(* IEC 61131-3 sources: YaoKangDeviceDemo/src/00_Globals, 6 files *)

(* ---- ST_StruHMI.st ---- *)
(*============================================================================
  HMI 线上结构体类型库 —— 寄存器布局契约
  ----------------------------------------------------------------------------
  权威来源：旧工程 InoProShop 变量表导出
    old/结构体/Stru_HMI_new.csv                     （主结构体，AT %MW200）
    old/结构体/Stru_HMI_DeviceInfo_new.csv          （设备信息镜像，AT %MW1000）
    old/结构体/Stru_HMI_DeviceIdentityWrite_new.csv （设备身份维护，AT %MW1010）

  ⚠ 铁律：类型名、字段名、字段顺序、数据类型、数组长度必须与 CSV 完全一致，
     一字不改。BOOL 按位打包、REAL/DINT 偶字对齐由编译器自动完成；
     本工程照抄定义并整体 AT 映射后，布局即与旧工程/HMI 完全相同。
  验收：下载后 InoProShop 变量表中 HMI 的 nBitLen 应 = 11856 bit（741 字，
        D200–D940），与旧工程一致。
==========================================================================*)

(*---------------------------------------------------------------------------
  通用命令：参数块统一操作集（Load/Apply/Save/ResetDefault + 回令）
  出现位置：Condition.ParamCmd / TailTilt.ConfigCmd / 3×Axis.ConfigCmd / HomingParams.Cmd
---------------------------------------------------------------------------*)
TYPE Stru_ConfigCmd :
STRUCT
    iErrorCode      : INT;      // 操作错误
    bLoad           : BOOL;     // 加载：从运行区读到缓冲区
    bApply          : BOOL;     // 应用：缓冲区覆盖运行区
    bSave           : BOOL;     // 保存：运行区写入 Retain
    bResetDefault   : BOOL;     // 恢复工厂默认
    bSuccess        : BOOL;     // 操作成功（PLC→HMI 回令）
    bError          : BOOL;     // 操作失败（只读，PLC→HMI 回令）
    bPad0           : BOOL;     // 填充
    bPad1           : BOOL;     // 对齐填充
END_STRUCT
END_TYPE

(*---------------------------------------------------------------------------
  调理区（Condition）
---------------------------------------------------------------------------*)
TYPE Stru_CondCmd :
STRUCT
    S1_StartProcess     : BOOL;     // 启动流程 (电平，CSV 注释；PLC 侧按 R_TRIG 消费亦安全)
    S2_StartChengJiao   : BOOL;     // 开始成角 (脉冲)
    S3_AllowSignal      : BOOL;     // 确认信号 (脉冲)
    bStop               : BOOL;     // 停止 (脉冲)
    bSignal             : BOOL;     // 脚踏信号 (脉冲/电平)
    bReset              : BOOL;     // 复位错误 (脉冲)
    bPause              : BOOL;     // 暂停
    bResume             : BOOL;     // 恢复
    bSkipAngle          : BOOL;     // 跳过成角 (脉冲, v3.16)
    bPpad               : BOOL[7];  // 填充（字段名照抄 CSV：bPpad）
END_STRUCT
END_TYPE

(* 单轴往复运动参数（SeatTwist / LegAngle / ChestImpact 三处复用） *)
TYPE Stru_ReciprocationSettings :
STRUCT
    arPosition      : REAL[16];    // 各段目标位置
    arVelocity      : REAL[16];    // 各段速度
    rAcc            : REAL;        // 加速度（必须 > 0）
    rDec            : REAL;        // 减速度（必须 > 0）
    rInitialPosition: REAL;        // 初始位置
    rReserved       : REAL;        // 保留
    iVelocityMode   : INT;         // 速度切换模式 0=独立速度 1=统一用 arVelocity[0]
    iCycleModeLen   : INT;         // 方向数组 abCycleMode 有效长度 (1~16)
    iCycleCount     : INT;         // 本轴循环次数，-1=用全局值
    iSignalMode     : INT;         // 本轴信号模式，-1=用全局值，0=点动 1=连动
    iSegmentCount   : INT;         // 运动段数 (1~16)，必须 >0 否则报错 1005
    iPadInt         : INT;         // 对齐填充
    bEnabled        : BOOL;        // 轴使能（FALSE=不参与联动，用于 2 轴场景）
    bOneWay         : BOOL;        // 单向还是多向
    abCycleMode     : BOOL[16];    // 方向数组
    bPad0           : BOOL;        // 填充
    bPad1           : BOOL;        // 对齐填充
END_STRUCT
END_TYPE

TYPE Stru_CondParams :
STRUCT
    SeatTwist       : Stru_ReciprocationSettings;   // 扭腰往复（线上顺序 Seat→Leg→Chest）
    LegAngle        : Stru_ReciprocationSettings;   // 摆腿往复
    ChestImpact     : Stru_ReciprocationSettings;   // 冲击往复
    rPusherPos      : REAL;        // 成角角度（尾板目标角度，度）
    rPusherInitPos   : REAL;        // 尾板初始角度
    diBatchCount    : DINT;        // 完整调理流程重复次数（老化模式）
    diBatchInterval : DINT;        // 批次间隔时间 (ms，老化模式)
    diTotalTimeout  : DINT;        // 总超时 (ms，默认 300000)
    diConfirmTimeout: DINT;        // HMI 等待确认超时 (ms，<=0=禁用)
    iCycleCount     : INT;         // 全局循环次数
    iSignalMode     : INT;         // 全局信号模式 (0=脚踏 1=自动)
END_STRUCT
END_TYPE

TYPE Stru_CondStatus :
STRUCT
    diActRunTime        : DINT;    // 实际运行时间 (ms，含暂停)
    diBatchCurrent      : DINT;    // 已完成批次数（老化）
    diBatchTarget       : DINT;    // 目标批次数（老化）
    diBatchRemainTime   : DINT;    // 批次间隔剩余时间 (ms)
    iPhase              : INT;     // 调理阶段 (0=空闲 1=预备 2=运行 3=成角 9=完成)
    iStep               : INT;     // 当前步骤（阶段内细分）
    iCurrentCycle       : INT;     // 当前循环次数
    iTargetCycles       : INT;     // 目标循环次数
    iErrorCode          : INT;     // 错误码
    iErrorLevel         : INT;     // 错误等级 0=L0 1=L1 2=L2
    iParamError         : INT;     // 参数验证错误码
    iParamErrorAxis     : INT;     // 参数错误所在轴 (1=Chest 2=Leg 3=Seat 4=Tail)
    iParamErrorField    : INT;     // 错误字段索引
    pad_int             : INT;     // 对齐填充
    bRunning            : BOOL;    // 调理进行中
    bDone               : BOOL;    // 调理已完成
    bPaused             : BOOL;    // 暂停中
    bError              : BOOL;    // 错误激活
    bBusy               : BOOL;    // 任意动作进行中
    bWaitingAngle       : BOOL;    // 等待成角
    bHoming             : BOOL;    // 回零中
    bAngleDone          : BOOL;    // 成角已完成
    bWaitingSignal      : BOOL;    // 等待脚踏信号
    bMoving             : BOOL;    // 往复动作中
    bHomeDone           : BOOL;    // 回零完成
    bManualStop         : BOOL;    // 手动停止
    bEmergencyStop      : BOOL;    // 紧急中止
    bParamValid         : BOOL;    // 参数校验通过
    bApplyDone          : BOOL;    // 参数应用完成
    bResetDone          : BOOL;    // 调理复位完成
    bBatchDone          : BOOL;    // 批量运行完成（老化）
END_STRUCT
END_TYPE

TYPE Stru_HMI_Condition :
STRUCT
    Cmd     : Stru_CondCmd;        // 调理命令
    Param   : Stru_CondParams;     // 调理参数（线上编辑区）
    Status  : Stru_CondStatus;     // 调理状态（PLC→HMI）
    ParamCmd: Stru_ConfigCmd;      // 参数块操作命令
END_STRUCT
END_TYPE

(*---------------------------------------------------------------------------
  系统区（Sys）
---------------------------------------------------------------------------*)
TYPE Stru_HMI_SysCmd :
STRUCT
    iWorkMode               : INT;
    iResetMode              : INT;
    iHomingMode             : INT;
    iUserRole               : INT;
    iAuthCode               : INT;
    arReservedInt           : INT[2];
    bServiceModeReq         : BOOL;
    bHomingReq              : BOOL;
    bStopReq                : BOOL;
    bPause                  : BOOL;
    bResume                 : BOOL;
    bAutoStartReq           : BOOL;
    bCalibrateReq           : BOOL;
    bResetReq               : BOOL;
    bAckErrorReq            : BOOL;
    bEmergencyStopReq       : BOOL;
    bInitializeReq          : BOOL;
    bServiceMechHomeReq     : BOOL;
    bSelfTestConfirm        : BOOL;
    bSelfTestSkip           : BOOL;
    bAllPowerOffReq         : BOOL;
    bAllPowerOnReq          : BOOL;
    bRevalidateParams       : BOOL;
    bServiceAuthConfirm     : BOOL;
    bNoLoadConfirm          : BOOL;
    bStartSelfTestReq       : BOOL;
    bServiceDoneReq         : BOOL;
    bReadyCheckReq          : BOOL;
    bQuickStartReq          : BOOL;
    bForceSkipSelfTestReq   : BOOL;
    bClearZeroRetainReq     : BOOL;
    bLearnImpactBiasReq     : BOOL;
    bPadHmi0                : BOOL;
END_STRUCT
END_TYPE

TYPE Stru_HMI_SysDisplay :
STRUCT
    rTailDriftPulse         : REAL;
    diUpTime                : DINT;
    diReadyCheckResult      : DINT;
    iState                  : INT;
    iPhase                  : INT;
    iInitErrorCode          : INT;
    iErrorCode              : INT;
    iErrorSubCode           : INT;
    iErrorLevel             : INT;
    iErrorSource            : INT;
    iHealthLevel            : INT;
    iTaskPhase              : INT;
    iBlockReason            : INT;
    iWorkMode               : INT;
    iPadInt                 : BOOL;     // CSV 中该字段类型为 BOOL，照抄
    bInitialized            : BOOL;
    bParamInitialized       : BOOL;
    bAutoProcessRunning     : BOOL;
    bPowerOn                : BOOL;
    bPoweringUp             : BOOL;
    bNeedReset              : BOOL;
    bTailSensorAtBoot       : BOOL;
    bHealthCheckSkipped     : BOOL;
    bAllAxesReferenced      : BOOL;
    bAllAxesHomed           : BOOL;
    bAllAxesAtInit          : BOOL;
    bAllAxesIdle            : BOOL;
    bAnyAxisAtLimit         : BOOL;
    bReady                  : BOOL;
    bSafeToStart            : BOOL;
    bBusy                   : BOOL;
    bParamError             : BOOL;
    bAbsPositionValid       : BOOL;
    bSensitiveRunning       : BOOL;
    bIsEmergency            : BOOL;
    bSelfTestDone           : BOOL;
    bSkipSelfTestAllowed    : BOOL;
    bForceSkipSelfTestAllowed: BOOL;
END_STRUCT
END_TYPE

TYPE Stru_ErrorEntry :
STRUCT
    iLevel      : INT;
    iCode       : INT;
    iSource     : INT;
    iVal1       : INT;
    diTimestamp : DINT;
END_STRUCT
END_TYPE

TYPE Stru_ErrorQueue :
STRUCT
    aEntries    : Stru_ErrorEntry[9];
    iHead       : INT;
    iTail       : INT;
    iCount      : INT;
    bOverflow   : BOOL;
    bPad0       : BOOL;
END_STRUCT
END_TYPE

TYPE Stru_HMI_SysRuntime :
STRUCT
    diAgingCycleCount   : DINT;
    diTotalCycles       : DINT;
    diRunTime           : DINT;
    diReserved          : DINT;
    iCurrentStep        : INT;
    iActCycles          : INT;
    bBatchDone          : BOOL;
    pad                 : BOOL;
END_STRUCT
END_TYPE

TYPE Stru_HMI_SysError :
STRUCT
    iLevel      : INT;
    iCode       : INT;
    iSource     : INT;
    iSubCode    : INT;
    iVal1       : INT;
    iVal2       : INT;
    bActive     : BOOL;
    bCritical   : BOOL;
    bEscalated  : BOOL;
    bNeedReset  : BOOL;
    pad0        : BOOL;
    pad1        : BOOL;
    pad2        : BOOL;
    pad3        : BOOL;
END_STRUCT
END_TYPE

TYPE Stru_HMI_SysWarning :
STRUCT
    iCode       : INT;
    iSource     : INT;
    iVal1       : INT;
    pad_int     : INT;
    bActive     : BOOL;
    pad0        : BOOL;
END_STRUCT
END_TYPE

TYPE Stru_HMI_Sys :
STRUCT
    Cmd         : Stru_HMI_SysCmd;
    Status      : Stru_HMI_SysDisplay;
    ErrorQueue  : Stru_ErrorQueue;
    Runtime     : Stru_HMI_SysRuntime;
    Error       : Stru_HMI_SysError;
    Warning     : Stru_HMI_SysWarning;
END_STRUCT
END_TYPE

(*---------------------------------------------------------------------------
  尾板/电推杆（TailTilt）
---------------------------------------------------------------------------*)
TYPE Stru_PusherCmd :
STRUCT
    bEnable         : BOOL;     // 使能
    bStop           : BOOL;     // 停止
    bReset          : BOOL;
    bCalibrate      : BOOL;     // 执行标定
    bAutoMove       : BOOL;     // 自动定位
    bHome           : BOOL;     // 回零（移动到原点位置）
    bJogUp          : BOOL;     // 正向点动
    bJogDown        : BOOL;     // 负向点动
    bManualPreset   : BOOL;     // 手动清零
    bResetError     : BOOL;     // 重置故障
    bPad            : BOOL[6];  // 填充
END_STRUCT
END_TYPE

TYPE Stru_PusherStatus :
STRUCT
    rCurrAngle              : REAL;     // 当前角度（HC_Counter mm 位置经余弦定理/ACOS 解算）
    rCurrPulse              : REAL;     // CSV 字段名照抄（原 AD/脉冲位置量）；本硬件无 AD，由 HC_Counter 位置(mm)镜像填入
    rPresetDeg              : REAL;     // 最近一次 Preset 目标角度
    rReserved               : REAL;
    iErrorCode              : INT;      // 错误码 (5001=堵转 5002=超时 5003=重试超限)
    iRetryCount             : INT;      // 当前重试计数
    bCalibrated             : BOOL;     // 已校准
    bHomed                  : BOOL;     // 已回零（Home 流程置位，与标定解耦）
    bHoming                 : BOOL;     // 正在执行 Home 流程
    bHomeSwitch             : BOOL;     // 原点传感器有效 (= I_Pusher_Origin)
    bReferenceValid         : BOOL;     // 坐标参考有效
    bHomeSensorHealthy      : BOOL;     // 原点传感器健康
    bHomeSensorStuckOn      : BOOL;     // 原点传感器卡死 ON
    bHomeSensorStuckOff     : BOOL;     // 原点传感器卡死 OFF/不可达
    bHomePlausible          : BOOL;     // 原点传感器与角度一致性通过
    bRunUp                  : BOOL;     // 正转输出
    bRunDown                : BOOL;     // 反转输出
    bBusy                   : BOOL;     // 忙
    bDone                   : BOOL;     // 完成
    bError                  : BOOL;     // 故障
    bWarning                : BOOL;
    bStall                  : BOOL;
    bTimeout                : BOOL;
    bPosLimit               : BOOL;
    bNegLimit               : BOOL;
    bAtInit                 : BOOL;
    bSensorChecked          : BOOL;     // 传感器已被检验（FB_Home.out_bSensorChecked 镜像）
    bAutoMovePending        : BOOL;
    bAutoMoveAllowed        : BOOL;
    bPadDiag0               : BOOL;
    bPadDiag1               : BOOL;
END_STRUCT
END_TYPE

TYPE Stru_PusherLimitConfig :
STRUCT
    rMaxDeg                 : REAL;     // 正限位 (°)
    rMinDeg                 : REAL;     // 负限位 (°)
    rTolerance              : REAL;     // 到位容差 (°，判断到位/bAtInit)
    rInitialPosition        : REAL;     // 初始位置角度 (°，回零目标)
    rMinTravel              : REAL;     // 最小行程保护 (°，堵转检测前必须走过)
    rHomePosition           : REAL;     // 原点位置 (°)
    rPulsePerDeg            : REAL;     // 脉冲当量 (Pulse/°)
    rAdOffset               : REAL;     // ★AD 字段保留不赋值：AD 零偏（无 AD 硬件，位置来自 HC_Counter）
    rAdScale                : REAL;     // ★AD 字段保留不赋值：AD 标度（无 AD 硬件）
    rFitK0                  : REAL;     // ★AD 字段保留不赋值：AD 拟合系数 K0（无 AD 硬件）
    rFitK1                  : REAL;     // ★AD 字段保留不赋值：AD 拟合系数 K1（无 AD 硬件）
    rFitK2                  : REAL;     // ★AD 字段保留不赋值：AD 拟合系数 K2（无 AD 硬件）
    rFitK3                  : REAL;     // ★AD 字段保留不赋值：AD 拟合系数 K3（无 AD 硬件）
    rAdJumpLimitDeg         : REAL;     // ★AD 字段保留不赋值：AD 跳变限幅 (°)（无 AD 硬件）
    rInertiaUp              : REAL;     // 角度增大方向惯性补偿 (°，提前停)
    rInertiaDown            : REAL;     // 角度减小方向惯性补偿 (°，提前停)
    rStallThreshold         : REAL;     // 堵转位移阈值 (°)
    rStallSpeedThreshold    : REAL;     // 堵转速度阈值 (°/s)
    diStallTimeout          : DINT;     // 堵转判定时间 (ms)
    diTimeout               : DINT;     // 寻传感器/标定超时 (ms)
    diReverseDelay          : DINT;     // 反向缓冲延时 (ms)
    diStopCheck             : DINT;     // 停车滑行等待 (ms)
    diAdMin                 : DINT;     // ★AD 字段保留不赋值：AD 采样下限原始码（无 AD 硬件）
    diAdMax                 : DINT;     // ★AD 字段保留不赋值：AD 采样上限原始码（无 AD 硬件）
    diAdSampleMs            : DINT;     // ★AD 字段保留不赋值：AD 采样周期 (ms)（无 AD 硬件）
    iMaxRetries             : INT;      // 最大修正次数
    iReferenceMode          : INT;      // ★AD 字段保留不赋值：参考模式 0=脉冲+HC 1=AD拟合（本硬件固定走 0，不写入）
    iPad                    : INT;      // 填充
    bInvertPusherDirection  : BOOL;     // 输出方向取反（Y5/Y6 交换，对齐物理方向）
END_STRUCT
END_TYPE

TYPE Stru_PusherMotion :
STRUCT
    rTargetAngle        : REAL;     // 目标角度 (°)
    rManualPresetAngle  : REAL;     // 手动 Preset 目标角度 (°)
    diJogTime           : DINT;     // Jog 限时 (ms，bJogModeTimed=TRUE 时生效)
    diMoveTimeout       : DINT;     // 定位超时 (ms)
    bJogModeTimed       : BOOL;     // 限时 Jog 模式
    bPad0               : BOOL;
END_STRUCT
END_TYPE

TYPE Stru_HMI_Pusher :
STRUCT
    Cmd         : Stru_PusherCmd;
    Status      : Stru_PusherStatus;
    ConfigCmd   : Stru_ConfigCmd;
    Config      : Stru_PusherLimitConfig;
    Motion      : Stru_PusherMotion;
END_STRUCT
END_TYPE

(*---------------------------------------------------------------------------
  伺服轴（ChestImpact / SeatTwist / LegAngle 三处复用）
  ⚠ 字段顺序照抄 CSV：Status → Cmd → Motion → Config → ConfigCmd
---------------------------------------------------------------------------*)
TYPE Stru_ServoAxisStatus :
STRUCT
    rActPosition            : REAL;     // 实际位置（脉冲或 mm）
    rActVelocity            : REAL;     // 实际速度
    rActTorque              : REAL;     // 实际扭矩
    iErrorCode              : INT;      // 错误码（来自 FB_运动控制）
    iDriveErrorCode         : INT;      // 驱动器错误码（来自伺服/M900）
    diDiscreteMotionTime    : DINT;     // 定位运动时间 (ms)
    bEnabled                : BOOL;     // 已使能（驱动器上电）
    bReady                  : BOOL;     // 驱动就绪
    bBusy                   : BOOL;     // 运动中
    bDone                   : BOOL;     // 动作完成（上升沿）
    bStandStill             : BOOL;     // 静止
    bInPosition             : BOOL;     // 到位
    bDiscreteMotion         : BOOL;     // 定位运动中
    bMoveDone               : BOOL;     // 运动完成 (脉冲)
    bZeroCommissioned       : BOOL;     // 底层 home-state 镜像（非持久建零标志）
    bZeroCommissioning      : BOOL;     // 正在原点标定（运行期通常不触发）
    bOriginSwitch           : BOOL;     // 原点传感器信号（物理输入）
    bPosLimit               : BOOL;     // 正限位触发
    bNegLimit               : BOOL;     // 负限位触发
    bError                  : BOOL;     // 错误激活
    bStopping               : BOOL;     // 错误停止中
    bEncoderFault           : BOOL;     // 编码器故障
    pad0                    : BOOL;
    pad1                    : BOOL;
    pad2                    : BOOL;
    bPad3                   : BOOL;     // CSV 中该字段名带 b 前缀，照抄
END_STRUCT
END_TYPE

TYPE Stru_AxisForceStatus :
STRUCT
    rBiasPosPct     : REAL;     // 正扭矩侧静止基线 (%)
    rBiasNegPct     : REAL;     // 负扭矩侧静止基线 (%)
    rNetTorquePct   : REAL;     // 扣基线后净扭矩 (%)
    rForceRawN      : REAL;     // 未滤波牵引力估算 (N)
    rForceFiltN     : REAL;     // 低通后牵引力估算 (N)
    diOverForceET   : DINT;     // 超力持续时间 (ms)
    bForceValid     : BOOL;     // 力估算有效
    bBiasPosValid   : BOOL;     // 正侧基线已学习
    bBiasNegValid   : BOOL;     // 负侧基线已学习
    bOverForce      : BOOL;     // 超力实时态
    bOverForceLatched: BOOL;    // 超力锁存
    bPad0           : BOOL;
END_STRUCT
END_TYPE

TYPE Stru_AxisStatus :
STRUCT
    Servo               : Stru_ServoAxisStatus;
    Force               : Stru_AxisForceStatus;
    iCurrentStep        : INT;      // 当前运动步骤 (0=空闲 1-N=执行中)
    iPadInt             : INT;      // 对齐填充
    diWaitingTime       : DINT;     // 等待时间 (ms)
    diMotionTime        : DINT;     // 运动用时 (ms)
    iErrorCode          : INT;      // [镜像] = Servo.iErrorCode
    bCalibrated         : BOOL;     // 已标定
    bError              : BOOL;
    bWarning            : BOOL;     // 警告激活（区别于 Servo.bError）
    bAxisErrorStopping  : BOOL;     // 轴错误停止中（区别于 Servo.bStopping）
    bAtInit             : BOOL;     // 在初始位置容差内
    bPad0               : BOOL;
END_STRUCT
END_TYPE

TYPE Stru_AxisCmd :
STRUCT
    bEnable             : BOOL;     // 使能（伺服上电）
    bReset              : BOOL;     // 复位（清除轴错误）
    bZeroCommission     : BOOL;     // 原点标定（仅工厂模式，触发 MC_Home，运行期禁止）
    bStop               : BOOL;     // 停止（立即减速停车）
    bMoveAbs            : BOOL;     // 绝对定位
    bMoveRel            : BOOL;     // 相对定位
    bJogPos             : BOOL;     // 正向点动（按住持续）
    bJogNeg             : BOOL;     // 负向点动（按住持续）
    bAutoMove           : BOOL;
    bMoveBuffer         : BOOL;
    bRequestDisable     : BOOL;     // 请求断使能（EMERGENCY_HOME 降级复位流程）
    bPad0               : BOOL;
    pad1                : BOOL;     // CSV 中该字段名无 b 前缀，照抄
    pad2                : BOOL;
    pad3                : BOOL;
    pad4                : BOOL;
END_STRUCT
END_TYPE

TYPE Stru_AxisMotionParam :
STRUCT
    rTargetPos  : REAL;     // 目标位置
    rTargetVel  : REAL;     // 目标速度
    rJogVel     : REAL;     // 点动速度
    rAcc        : REAL;     // 加速度
    rDec        : REAL;     // 减速度
    rInitPos    : REAL;     // 初始位置
    diTimeout   : DINT;     // 超时 (ms)
    rReserved   : REAL;
END_STRUCT
END_TYPE

TYPE Stru_AxisLimitConfig :
STRUCT
    rPosLimit       : REAL;     // 正限位 (°或 mm)
    rNegLimit       : REAL;     // 负限位 (°或 mm)
    rInitPos        : REAL;     // 初始位置
    rTolerance      : REAL;     // 到位容差 (°或 mm)
    rMaxVel         : REAL;     // 最大速度
    rMinVel         : REAL;     // 最小速度
    rMaxAcc         : REAL;     // 最大加速度
    rMaxDec         : REAL;     // 最大减速度
    diPulsePerDeg   : DINT;     // 脉冲当量 (Pulse/°)
    diTimeout       : DINT;     // 超时报警 (ms)
END_STRUCT
END_TYPE

TYPE Stru_HMI_Axis :
STRUCT
    Status      : Stru_AxisStatus;
    Cmd         : Stru_AxisCmd;
    Motion      : Stru_AxisMotionParam;
    Config      : Stru_AxisLimitConfig;
    ConfigCmd   : Stru_ConfigCmd;
END_STRUCT
END_TYPE

(*---------------------------------------------------------------------------
  回零参数（HomingParams）
---------------------------------------------------------------------------*)
TYPE Stru_HomingParams :
STRUCT
    rLimitEscapeVel         : REAL;
    rChestJogVel            : REAL;
    rLegJogVel              : REAL;
    rSeatJogVel             : REAL;
    rChestCrawlVel          : REAL;
    rLegCrawlVel            : REAL;
    rSeatCrawlVel           : REAL;
    rChestApproachZone      : REAL;
    rLegApproachZone        : REAL;
    rSeatApproachZone       : REAL;
    rChestHysteresis        : REAL;
    rLegHysteresis          : REAL;
    rSeatHysteresis         : REAL;
    rChestJogAcc            : REAL;
    rLegJogAcc              : REAL;
    rSeatJogAcc             : REAL;
    rAntiPinchTorqueLimit   : REAL;
    diHomingTimeout         : DINT;
    diEmergencyTimeout      : DINT;
    diLimitEscapeTimeout    : DINT;
    diStopReleaseTimeout    : DINT;
    diEmergencyCoastMs      : DINT;
    diEmergencyStallTimeout : DINT;
    iHomingMode             : INT;
    iMaxRetry               : INT;
    bEmergencyAllowCalib    : BOOL;
    bPad0                   : BOOL;
END_STRUCT
END_TYPE

TYPE Stru_HMI_HomingParams :
STRUCT
    Cmd     : Stru_ConfigCmd;
    Params  : Stru_HomingParams;
END_STRUCT
END_TYPE

(*---------------------------------------------------------------------------
  尾板位置/角度反馈（D936–D940，不挤占 TailTilt 主协议）
  字段名照抄 CSV（原为 AD 拟合反馈窗：拟合角/AD原始值/AD有效位）。
  真实硬件无 AD：位置来自 HC_Counter(mm)、角度由几何解算——rAdAngle 填几何解算
  角度、bAdValid 填 HC_Counter 有效位；diAdRaw（AD 原始码）无对应物理量，
  保持 0 不赋值；布局 5 字不变。
---------------------------------------------------------------------------*)
TYPE Stru_HMI_TailAdFeedback :
STRUCT
    rAdAngle    : REAL;     // 字段名照抄 CSV（AD 拟合角）；本硬件填几何解算角度（°，D936–D937）
    diAdRaw     : DINT;     // ★AD 字段保留不赋值：AD 原始码（无 AD 硬件，保持 0，D938–D939）
    bAdValid    : BOOL;     // 字段名照抄 CSV（AD 有效位）；本硬件填 HC_Counter.Valid 且无 Error
    bPad0       : BOOL;     // 填充
END_STRUCT
END_TYPE

(*---------------------------------------------------------------------------
  主结构体：HMI，整体 AT %MW200（D200–D940，741 字）
  ⚠ 成员顺序照抄 CSV：Condition / Sys / TailTilt / ChestImpact / SeatTwist /
     LegAngle / HomingParams / TailTiltAdFeedback
---------------------------------------------------------------------------*)
TYPE Stru_HMI :
STRUCT
    Condition           : Stru_HMI_Condition;      // 调理参数、控制、状态
    Sys                 : Stru_HMI_Sys;            // 系统
    TailTilt            : Stru_HMI_Pusher;         // 尾板下降（电推杆）
    ChestImpact         : Stru_HMI_Axis;           // 冲击轴
    SeatTwist           : Stru_HMI_Axis;           // 扭角轴
    LegAngle            : Stru_HMI_Axis;           // 转角轴
    HomingParams        : Stru_HMI_HomingParams;   // 回零参数
    TailTiltAdFeedback  : Stru_HMI_TailAdFeedback; // 尾板位置/角度反馈（D936–D940，mm+几何角度）
END_STRUCT
END_TYPE

(*---------------------------------------------------------------------------
  设备信息只读镜像（D1000–D1004）—— Stru_HMI_DeviceInfo_new.csv
---------------------------------------------------------------------------*)
TYPE Stru_HMI_DeviceInfo :
STRUCT
    diDeviceNoRaw   : DINT;     // 原始设备编号（工厂烧录/维护配置）
    iMacWord0       : INT;      // PLC MAC 地址字 0 (= _Ethernet.MACAddress[0])
    iMacWord1       : INT;      // PLC MAC 地址字 1 (= _Ethernet.MACAddress[1])
    iMacWord2       : INT;      // PLC MAC 地址字 2 (= _Ethernet.MACAddress[2])
END_STRUCT
END_TYPE

(*---------------------------------------------------------------------------
  设备身份维护写入（D1010–D1013）—— Stru_HMI_DeviceIdentityWrite_new.csv
  例外：本块命令集仅 Load / Apply（无 Save / ResetDefault）
---------------------------------------------------------------------------*)
TYPE Stru_DeviceIdentityCmd :
STRUCT
    iErrorCode  : INT;
    bLoad       : BOOL;
    bApply      : BOOL;
    bSuccess    : BOOL;
    bError      : BOOL;
    bPad0       : BOOL;
    bPad1       : BOOL;
END_STRUCT
END_TYPE

TYPE Stru_HMI_DeviceIdentityWrite :
STRUCT
    Cmd             : Stru_DeviceIdentityCmd;
    diDeviceNoRaw   : DINT;     // DINT 偶字对齐 → D1012–D1013
END_STRUCT
END_TYPE

(* ---- GVL_CONST.st ---- *)
(*============================================================================
  常量库：状态码 / 错误码 / 角色 / 轴索引
  禁止魔法数字；新增码值须与《HMI-PLC地址分配表.md》对齐。
==========================================================================*)

VAR_GLOBAL CONSTANT
    (*--- 主状态 iState（MODE_MANAGER，13 态） ---*)
    ST_INIT              : INT := 0;
    ST_READY_CHECK       : INT := 3;
    ST_SELFTEST          : INT := 5;
    ST_STANDBY           : INT := 10;
    ST_SERVICE_REQUIRED  : INT := 15;
    ST_AUTORUN           : INT := 20;
    ST_SERVICE           : INT := 30;
    ST_HOMING            : INT := 40;
    ST_CALIBRATE         : INT := 45;
    ST_RESET             : INT := 50;
    ST_STOPPING          : INT := 60;
    ST_SOFT_ESTOP        : INT := 110;
    ST_HARD_ESTOP        : INT := 120;
    ST_PARAM_LIMITED     : INT := 998;

    (*--- 调理阶段 iPhase（Condition.Status.iPhase） ---*)
    COND_IDLE            : INT := 0;
    COND_PREPARE         : INT := 1;
    COND_RUNNING         : INT := 2;
    COND_ANGLE           : INT := 3;
    COND_DONE            : INT := 9;

    (*--- 工作模式 ---*)
    WORKMODE_COND        : INT := 1;    (* 调理 *)
    WORKMODE_TREAT       : INT := 2;    (* 治疗 *)
    WORKMODE_AGING       : INT := 3;    (* 老化 *)

    (*--- 用户角色（HMI 线协议：0=操作员 1=工程师；退出登录/未登录=操作员 0） ---*)
    ROLE_NONE            : INT := 0;
    ROLE_OPERATOR        : INT := 0;
    ROLE_ENGINEER        : INT := 1;
    AUTH_CODE_ENGINEER   : INT := 16#5A;   (* 登录写 16#5A、退出写 0（防误写） *)

    (*--- 轴索引（故障来源 gFaultSource / 参数错误上报用，INT 编号） ---*)
    (* 注：勿与 GVL_IoMap 中 Axis_胸背/臀盘/臀腿（AXIS_REF 轴引用）混淆，
       ST 标识符大小写不敏感，故本组常量使用 AXIS_ID_ 前缀。 *)
    AXIS_ID_CHEST        : INT := 1;    (* 冲击 *)
    AXIS_ID_LEG          : INT := 2;    (* 转角 *)
    AXIS_ID_SEAT         : INT := 3;    (* 扭角 *)
    AXIS_ID_TAIL         : INT := 4;    (* 尾板推杆 *)

    (*--- 错误码段位约定：
       1xxx 系统/急停  11xx 初始化/电源  12xx 紧急回零/防夹/跟随  13xx 自检
       2xxx 三轴       3xxx 推杆(3021-3025/3101-3107)  4xxx 回零
       45xx 阻塞原因(iBlockReason,MODE_MANAGER 写,HMI 显示"当前活跃任务阶段与阻塞原因")
       5xxx 参数/身份(5001-5003/5005/5006)                          7xxx 调理前检查
       子码约定：轴故障 iSubCode=驱动器 Er.xxx；gFaultSource 用 AXIS_ID_* / SRC_*。
       级别：1001/1002/1003 段码由 ERROR_MANAGER 按码表定级（Critical 需手动复位）。 ---*)

    (*===== 1xxx 系统 / 急停 =====*)
    ERR_HARD_ESTOP       : INT := 1001;   (* 硬急停：物理急停链路断开（常闭点断开/安全继电器动作） *)
    ERR_SOFT_ESTOP       : INT := 1002;   (* 软急停：HMI 急停请求（D488.9，受控减速） *)
    ERR_ESTOP_MISMATCH   : INT := 1003;   (* 急停双通道不一致（通道1/通道2 状态分歧） *)
    ERR_SOFT_ESTOP_TOUT  : INT := 1004;   (* 软急停减速超时，升级硬急停 *)
    ERR_COMM_LOST        : INT := 1006;   (* HMI 通信超时（Modbus 心跳丢失） *)
    ERR_SCAN_WATCHDOG    : INT := 1007;   (* 扫描周期看门狗超时 *)

    (*===== 11xx 初始化 / 电源 =====*)
    ERR_INIT_POWER       : INT := 1101;   (* 伺服上电失败（使能超时无 bReady） *)
    ERR_INIT_AXIS_REF    : INT := 1102;   (* 轴参考/零点标志丢失，需回零 *)
    ERR_INIT_CONFIG      : INT := 1103;   (* 启动参数未应用/配置无效 *)

    (*===== 12xx 紧急回零 / 防夹 / 跟随 =====*)
    ERR_EMGHOME_RELEASE  : INT := 1201;   (* 紧急回零：MC_Stop 释放等待超时 *)
    ERR_EMGHOME_TORQUE   : INT := 1202;   (* 紧急回零：扭矩防夹触发（超阈重试上限内） *)
    ERR_EMGHOME_RETRY    : INT := 1203;   (* 紧急回零：防夹重试超限，中止 *)
    ERR_ANTIPINCH_JOG    : INT := 1204;   (* Jog 防夹：点动扭矩超阈，立即停止 *)
    ERR_AXIS_FOLLOW      : INT := 1205;   (* 跟随误差超限（位置偏差过大） *)
    ERR_OVERFORCE        : INT := 1206;   (* 超力保护：牵引力估算超阈持续超时，锁存停机 *)

    (*===== 13xx 自检 =====*)
    ERR_SELFTEST_ENTRY   : INT := 1301;   (* 自检门禁断言不满足 *)
    ERR_SELFTEST_TIMEOUT : INT := 1302;   (* 自检全局超时 *)
    ERR_SELFTEST_PUSHER  : INT := 1303;   (* 自检推杆参考/校准失败（30s 超时） *)
    ERR_SELFTEST_AXIS    : INT := 1304;   (* 自检三轴 ±2° 单循环失败（8s/轴超时） *)
    ERR_SELFTEST_DIRTY   : INT := 1305;   (* 自检完成后脏标记未清零 *)

    (*===== 2xxx 三轴伺服 =====*)
    ERR_AXIS_DRIVE       : INT := 2001;   (* 驱动器故障（子码=驱动器 Er.xxx） *)
    ERR_AXIS_ENCODER     : INT := 2002;   (* 编码器故障，绝对位置不可信，禁定位 *)
    ERR_AXIS_HWLIMIT     : INT := 2003;   (* 硬限位触发 *)
    ERR_AXIS_SWLIMIT     : INT := 2004;   (* 软限位：越限运动被禁 *)
    ERR_AXIS_STEP_TOUT   : INT := 2005;   (* 运动步骤超时（目标未在 diTimeout 内到达） *)
    ERR_AXIS_CMD_ILLEGAL : INT := 2006;   (* 轴命令非法（未使能/未参考时请求定位） *)

    (*===== 3xxx 电推杆（尾板成角） =====*)
    ERR_TAIL_SENSOR_STKON  : INT := 3021; (* 原点传感器卡死 ON（应断开通） *)
    ERR_TAIL_SENSOR_STKOFF : INT := 3022; (* 原点传感器卡死 OFF（应接通通不了） *)
    ERR_TAIL_SENSOR_IMPL   : INT := 3023; (* 原点与角度一致性不合理（参考冲突） *)
    ERR_TAIL_NOT_CALIB     : INT := 3024; (* 未校准/参考无效，禁止自动定位 *)
    ERR_TAIL_ANGLE_LIMIT   : INT := 3025; (* 角度软限位保护动作 *)
    ERR_TAIL_CAL_TOP       : INT := 3101; (* 校准：上行撞顶堵转 *)
    ERR_TAIL_CAL_HOME      : INT := 3102; (* 校准：上行找原点失败 *)
    ERR_TAIL_CAL_ESCAPE    : INT := 3103; (* 校准：下行脱离原点失败 *)
    ERR_TAIL_CAL_DEBOUNCE  : INT := 3104; (* 校准：原点去抖 30ms 不稳定 *)
    ERR_TAIL_CAL_TIMEOUT   : INT := 3105; (* 校准：全局超时 *)
    ERR_TAIL_CAL_DIR       : INT := 3106; (* 校准：方向逻辑异常（上下行判断矛盾） *)
    ERR_TAIL_HOME_FAILED   : INT := 3107; (* 回零失败 *)

    (*===== 4xxx 回零 =====*)
    ERR_HOME_TIMEOUT     : INT := 4001;   (* 普通回零全流程超时 *)
    ERR_HOME_REFUSE      : INT := 4002;   (* 回零被拒（安全/参考条件不满足） *)
    ERR_HOME_AXIS        : INT := 4003;   (* 某轴回初始位失败（子码=轴号） *)

    (*===== 45xx 阻塞原因（iBlockReason，MODE_MANAGER 唯一写，HMI 显示"当前活跃任务阶段与阻塞原因"）
       0=无阻塞；>0 时 HMI 置灰启动/权限入口并提示。原因码为"就绪态最新阻塞"，
       与 diReadyCheckResult 位掩码并行：掩码供调试，原因码供界面直接显示。 =====*)
    BLOCK_REASON_SAFETY  : INT := 4501;   (* 安全链动作（硬/软急停或保护停机中） *)
    BLOCK_REASON_FAULT   : INT := 4502;   (* 存在活动 Critical 故障，需复位 *)
    BLOCK_REASON_AUTH    : INT := 4503;   (* 权限不足（维护/标定/自检需工程师角色+权限码 16#5A） *)
    BLOCK_REASON_POWER   : INT := 4504;   (* 硬件未上电/伺服未就绪 *)
    BLOCK_REASON_ZERO    : INT := 4505;   (* 未建零（三轴/推杆零点未标定，需维护建零） *)
    BLOCK_REASON_PARAM   : INT := 4506;   (* 运行参数无效（参数区未装载或校验未过） *)
    BLOCK_REASON_REF     : INT := 4507;   (* 轴参考无效（未回零/参考丢失） *)
    BLOCK_REASON_POS     : INT := 4508;   (* 未在初始位（轴当前位置偏离初始位，需回零） *)
    BLOCK_REASON_BUSY    : INT := 4509;   (* 系统忙（自动/自检/回零/标定等任务进行中） *)

    (*===== 5xxx 参数 / 身份 =====*)
    ERR_PARAM_LOCKED        : INT := 5004;   (* 参数 Apply/ResetDefault 被拒：自动流程运行中，运行区快照锁定 *)
    ERR_PARAM_DEVICE_LOCKED : INT := 5005;   (* 设备身份写入：锁定/状态不允许 *)
    ERR_PARAM_DEVICE_VALUE  : INT := 5006;   (* 设备编号非法 *)
    ERR_PARAM_VALUE         : INT := 5007;   (* 参数值非法（越界/≤0/逻辑矛盾），三元组定位到轴+字段 *)

    (*--- READY_CHECK 六项资格位掩码（Sys.Status.diReadyCheckResult，0=全过，置位=缺项） ---*)
    READY_BIT_ZERO    : INT := 0;   (* bit0：零点/参考无效（未建零或未回零） *)
    READY_BIT_PARAM   : INT := 1;   (* bit1：运行区参数无效/参数校验未过 *)
    READY_BIT_HW      : INT := 2;   (* bit2：硬件未就绪（未上电/伺服未使能） *)
    READY_BIT_HEALTH  : INT := 3;   (* bit3：健康检查未过（活动 Critical 错误） *)
    READY_BIT_POS     : INT := 4;   (* bit4：全轴未在初始位 *)
    READY_BIT_REF     : INT := 5;   (* bit5：全轴参考无效 *)

    (*--- 健康等级 iHealthLevel（Sys.Status） ---*)
    HEALTH_FAULT   : INT := 0;   (* 故障：有活动 Critical，禁止运行 *)
    HEALTH_NORMAL  : INT := 1;   (* 正常：全部资格具备 *)
    HEALTH_WARNING : INT := 2;   (* 警告：有活动 Warning，允许运行 *)
    HEALTH_UNKNOWN : INT := 3;   (* 未就绪：未完成自检/就绪检查 *)

    (*--- 电推杆错误码（TailTilt.Status.iErrorCode，业务码） ---*)
    PUSHER_ERR_STALL     : INT := 5001;  (* 堵转 *)
    PUSHER_ERR_TIMEOUT   : INT := 5002;  (* 超时 *)
    PUSHER_ERR_RETRY     : INT := 5003;  (* 重试超限 *)

    (*--- 参数校验错误（Condition.Status） ---*)
    PARAM_ERR_SEGMENT    : INT := 1005;  (* iSegmentCount 非法（校验类，Warning） *)

    (*===== 7xxx 调理前检查 / 运行条件 =====*)
    ERR_PRECHK_READY     : INT := 7001;   (* 就绪检查未通过（资格位掩码见 diReadyCheckResult） *)
    ERR_PRECHK_AXIS      : INT := 7002;   (* 启动前检查：轴未使能/未静止 *)
    ERR_PRECHK_POS        : INT := 7003;  (* 启动前检查：全轴未在初始位 *)
    ERR_PRECHK_PARAM     : INT := 7004;   (* 启动前检查：参数校验未通过 *)
    ERR_PRECHK_ZERO      : INT := 7005;   (* 启动前检查：零点/参考无效 *)

    (*--- 故障来源模块码 gFaultSource（轴用 AXIS_ID_CHEST/LEG/SEAT/TAIL=1..4） ---*)
    SRC_SAFETY           : INT := 10;   (* SAFETY_MANAGER *)
    SRC_MODE             : INT := 11;   (* MODE_MANAGER *)
    SRC_PARAM            : INT := 12;   (* PARAM_SERVICE *)
    SRC_MONITOR          : INT := 13;   (* MONITOR / AD / 通信 *)
    SRC_POWER            : INT := 14;   (* POWER *)
    SRC_OUTPUT           : INT := 15;   (* OUTPUT_ADAPTER（三轴） *)
    SRC_HOMING           : INT := 16;   (* 回零/紧急回零任务 *)
    SRC_SELFTEST         : INT := 17;   (* 自检任务 *)
    SRC_COND             : INT := 18;   (* 调理/治疗/老化任务 *)
    SRC_PUSHER           : INT := 19;   (* 推杆任务（区别于轴来源 AXIS_ID_TAIL=4） *)

    (*--- 轴命令位索引（Gvl.axisPulse / axisPulse 等 [3×N] 数组第二维下标）
       与 Stru_AxisCmd 中"脉冲型"字段一一对应；bJogPos/bJogNeg 为电平型，
       单独走 axisJogPos/axisJogNeg 镜像数组，不在本索引内。 ---*)
    AXCMD_RESET          : INT := 1;   (* bReset 复位清错 *)
    AXCMD_ZERO_COMM      : INT := 2;   (* bZeroCommission 原点标定（工厂） *)
    AXCMD_STOP           : INT := 3;   (* bStop 立即减速停车 *)
    AXCMD_MOVEABS        : INT := 4;   (* bMoveAbs 绝对定位 *)
    AXCMD_MOVEREL        : INT := 5;   (* bMoveRel 相对定位 *)
    AXCMD_AUTOMOVE       : INT := 6;   (* bAutoMove 自动流程运动 *)
    AXCMD_MOVEBUFFER     : INT := 7;   (* bMoveBuffer 16 段缓冲 *)
    AXCMD_REQ_DISABLE    : INT := 8;   (* bRequestDisable 请求断使能 *)
    AXCMD_MAX            : INT := 8;   (* 脉冲命令位个数（数组下界基准） *)

    (*--- FB_AxisControl 运动状态机步号（iStep / stStatus.iCurrentStep） ---*)
    AXST_IDLE            : INT := 0;   (* 未使能 *)
    AXST_ENABLING        : INT := 1;   (* 使能中 *)
    AXST_READY           : INT := 2;   (* 已使能静止就绪 *)
    AXST_JOG             : INT := 3;   (* 点动中 *)
    AXST_MOVE            : INT := 4;   (* 单段定位中 *)
    AXST_BUFFER          : INT := 5;   (* 多段缓冲执行中 *)
    AXST_ERROR           : INT := 9;   (* 轴错误态（驱动器故障/超时） *)

    (*--- POWER 分时上电时序（按 10ms 扫描周期推算，任务组态确认后统一修正） ---*)
    SCAN_PERIOD_MS      : DINT := 10;     (* 主任务扫描周期 (ms)，任务组态确认后统一修正；diMsTick 累加基准 *)
    PWR_STAGGER_SCAN    : DINT := 50;     (* 逐轴使能间隔扫描数（50 扫≈500ms，防浪涌） *)
    PWR_ENABLE_TIMEOUT  : DINT := 300;    (* 单轴使能确认超时扫描数（300 扫≈3s，超时报 1101） *)

    (*--- 力估算占位常量（台架标定 TODO：换算系数/阈值/持续时间需实测标定） ---*)
    FORCE_LPF_ALPHA      : REAL := 0.1;    (* 牵引力一阶低通系数（每扫 0.1，@10ms） *)
    FORCE_SCALE_N        : REAL := 1.0;    (* 净扭矩% → 牵引力 N 换算系数（占位） *)
    OVERFORCE_N          : REAL := 100.0;  (* 超力阈值 N（低通后，占位） *)
    OVERFORCE_SCAN       : DINT := 50;     (* 超力持续扫描数（50 扫≈500ms@10ms）锁存 *)

    (*===== P9 任务步号（TASK_RUNNER 写 Condition.Status.iStep / iPhase；
           CASE 标签仍用字面整数 + 行尾注释，本处仅为消除魔法数字。 =====*)

    (*--- 普通回零（iState=ST_HOMING=40）：三轴 MoveAbs 回 rInitPos ---*)
    HOMSEQ_START         : INT := 4000;   (* 入口：装载目标/启动快照 *)
    HOMSEQ_MOVE          : INT := 4010;   (* 发 MoveAbs（顺序模式逐轴 / 并行模式全发） *)
    HOMSEQ_WAIT          : INT := 4020;   (* 等待全轴到位（4001 全流程超时） *)
    HOMSEQ_DONE          : INT := 4090;   (* 完成：置参考有效/位标志，iPhase=COND_DONE *)

    (*--- 回零执行模式（runHoming.iHomingMode） ---*)
    HOM_MODE_SEQUENTIAL  : INT := 0;      (* 顺序：Chest→Seat→Leg 逐轴 *)
    HOM_MODE_PARALLEL    : INT := 1;      (* 并行：三轴同时 MoveAbs *)

    (*--- 紧急回零（iState=ST_SOFT_ESTOP=110 内）：四段 Jog 回初始位 + 防夹 ---*)
    EMH_WAIT_RELEASE     : INT := 1100;   (* 等 MC_Stop 释放/停稳（1201 diStopReleaseTimeout） *)
    EMH_JOG_MAIN         : INT := 1110;   (* 主速 Jog 回初始位（超接近区前） *)
    EMH_JOG_CRAWL        : INT := 1120;   (* 爬行 Jog（进入 rApproachZone 后） *)
    EMH_SETTLE           : INT := 1130;   (* 微调/迟滞判停（|pos-init|<=rHysteresis） *)
    EMH_PINCH_WAIT       : INT := 1140;   (* 防夹触发后撤力等待（1202，重试计数） *)
    EMH_DONE             : INT := 1190;   (* 紧急回零完成（停车电平保持，等 trigSysReset） *)

    (*--- 动态自检（iState=ST_SELFTEST=5）：Step10 → 100 成功 / 200 失败 ---*)
    ST_GATE              : INT := 10;     (* 门禁断言（1301） *)
    ST_WAIT_CONFIRM      : INT := 20;     (* 等安全确认（可跳过/工程师强跳） *)
    ST_PUSHER_CALIB      : INT := 30;     (* 推杆参考检查 + 校准（1303，30s） *)
    ST_ANGLE             : INT := 40;     (* 成角（推杆自动定位到自检角） *)
    ST_AXIS_CYCLE        : INT := 50;     (* 三轴 ±2° 单循环（1304，8s/轴） *)
    ST_ANGLE_RETURN      : INT := 60;     (* 成角回零（推杆回零/回初始角） *)
    ST_DIRTY_CHECK       : INT := 70;     (* 清/核四个脏标记（1305） *)
    ST_STEP_DONE         : INT := 100;    (* 自检成功（bSelfTestDone:=TRUE） *)
    ST_STEP_FAIL         : INT := 200;    (* 自检失败（Critical 上报，等复位） *)

    (*--- 维护建零（iState=ST_CALIBRATE=45）：6 重门控 ---*)
    CAL_GATE             : INT := 5000;   (* 6 重门控断言（工程师/授权/空载/静止/安全/参考） *)
    CAL_COMM             : INT := 5010;   (* 发三轴 AXCMD_ZERO_COMM + 推杆标定脉冲 *)
    CAL_CONFIRM          : INT := 5020;   (* 等 Retain 握手回读（bZeroCommSetReq/bPushCalibDoneLatch） *)
    CAL_DONE             : INT := 5090;   (* 建零完成，iPhase=COND_DONE *)

    (*--- 自检运动参数（占位常量，与计划 ±2°/8s 对齐） ---*)
    ST_SWING_DEG         : REAL := 2.0;   (* 单循环摆动幅度 ±2°（相对 rInitPos） *)
    ST_AXIS_TOUT_SCAN    : DINT := 800;   (* 单轴单循环超时 800 扫 ≈ 8s（1304） *)
    ST_PUSHER_TOUT_SCAN  : DINT := 3000;  (* 推杆校准超时 3000 扫 ≈ 30s（1303） *)
    ST_GLOBAL_TOUT_SCAN  : DINT := 12000; (* 自检全局超时 12000 扫 ≈ 120s（1302） *)
    ST_ANGLE_DEG         : REAL := 15.0;  (* 自检成角目标（占位，取推杆配置安全角） *)

    (*===== P10 调理/治疗/老化任务步号（iState=ST_AUTORUN=20 内 iStepCond，
           写 Condition.Status.iStep；CASE 标签仍用字面整数 + 行尾注释。 =====*)
    CONDSEQ_GATE         : INT := 105;    (* 启动前检查（急停/就绪/参考/初始位/使能/参数，7001-7005） *)
    CONDSEQ_WAIT_PREP    : INT := 108;    (* 等待人员准备（S2 成角 / 跳过成角） *)
    CONDSEQ_ANGLE        : INT := 110;    (* 成角定位（推杆 AutoMove → rPusherPos） *)
    CONDSEQ_WAIT_SIGNAL  : INT := 120;    (* 等待开始确认（S3/脚踏；信号模式=1 自动放行） *)
    CONDSEQ_RUN          : INT := 130;    (* 三轴 16 段轨迹 × 循环联动（暂停/恢复贯穿） *)
    CONDSEQ_LAND         : INT := 140;    (* 安全降落（推杆回 rPusherInitPos，bDone 判定） *)
    CONDSEQ_BATCH_WAIT   : INT := 145;    (* 老化批间等待（diBatchInterval，批次进度上报） *)
    CONDSEQ_DONE         : INT := 800;    (* 完成（bDone，iPhase=COND_DONE） *)
    CONDSEQ_FAIL         : INT := 900;    (* 异常收口（bError；急停/手动停止由 ModeManager 转态） *)

    (*--- 停止安全降落步号（iState=ST_STOPPING=60 内 iStepStop） ---*)
    STOPSEQ_HALT         : INT := 6000;   (* 发三轴 STOP 脉冲至全轴静止 *)
    STOPSEQ_RETURN       : INT := 6010;   (* 三轴并行 MoveAbs 回初始位（到位后 ModeManager 回 STANDBY） *)

    (*===== 7xxx 补充：调理运行期超时（7001-7005 见前） =====*)
    ERR_COND_RUN_TIMEOUT : INT := 7006;   (* 调理流程总超时（diTotalTimeout，单批） *)
    ERR_COND_CONFIRM_TOUT: INT := 7007;   (* 等待人员准备/开始确认超时（diConfirmTimeout，Warning） *)

    (*===== 尾板推杆几何解算固定常量（真实推杆：开关型电推杆 + HC_Counter 读 mm 位置，
           余弦定理/ACOS 解算当前角度；无 AD。算法蓝本：推杆轴控制方式.txt。
           ★ 下列长度/补偿均为机械几何量，现场实测标定后固化，禁止运行时修改。 =====*)
    PUSHER_GEO_VERT_MM   : REAL := 100.0; (* 旋转中心垂直长度（mm，占位待实测） *)
    PUSHER_GEO_PAR_MM    : REAL := 100.0; (* 旋转中心平行长度（mm，占位待实测） *)
    PUSHER_GEO_TILT0_MM  : REAL := 100.0; (* 旋转中心倾斜长度零位偏置（mm，占位待实测）；
                                             倾斜长度_1 = 本偏置 + 当前推杆位置(mm)，钳 >=0 *)
    PUSHER_GEO_FIX_ANG   : REAL := 72.6;  (* 固定角（°）：当前角度 = 180 - 72.6 - ACOS·180/π + 补偿 *)
    PUSHER_GEO_ANG_COMP  : REAL := 0.0;   (* 角度补偿（°，占位待实测） *)
    PUSHER_PI            : REAL := 3.14159; (* 圆周率（弧度→度换算，ACOS 输出为弧度） *)
END_VAR

(* ---- GVL_HMI.st ---- *)
(*============================================================================
  HMI 寄存器映射全局变量（D 区 / %MW）
  ----------------------------------------------------------------------------
  变量名 : 结构体类型           地址          范围           方向
    HMI                      Stru_HMI                     AT %MW200   D200–D940    双向
    HMI_DeviceIdentity       Stru_HMI_DeviceInfo          AT %MW1000  D1000–D1004  PLC→HMI 只读
    HMI_DeviceIdentityWrite  Stru_HMI_DeviceIdentityWrite AT %MW1010  D1010–D1013  双向

  注：变量名与类型名同名（用户指定）。
  HMI 为旧工程导出的主结构体，nBitLen=11856 bit = 741 字，下载后须核对
  InoProShop 变量表中 HMI 长度与基址与旧工程一致。
==========================================================================*)
VAR_GLOBAL
    HMI                     : Stru_HMI                     AT %MW200;   (* D200–D940  *)
    HMI_DeviceIdentity      : Stru_HMI_DeviceInfo          AT %MW1000;  (* D1000–D1004 *)
    HMI_DeviceIdentityWrite : Stru_HMI_DeviceIdentityWrite AT %MW1010;  (* D1010–D1013 *)
END_VAR

(* ---- GVL_Internal.st ---- *)
(*============================================================================
  内部全局变量（不映射 D 区，层间通信）
  ----------------------------------------------------------------------------
  单写源硬约束（见开发计划 §0.4）：
    iState / iWorkMode ......... MODE_MANAGER 唯一写
    Error / Warning / Queue .... ERROR_MANAGER 唯一写
    轴 bEnable / MC 指令 ....... POWER / OUTPUT_ADAPTER 唯一写
    任务级请求 ................. 各任务模块经 gTrig* / FaultReq 提交
==========================================================================*)
VAR_GLOBAL
    (*--- 系统状态（MODE_MANAGER 单写） ---*)
    iState          : INT := 0;        (* 主状态码，见 GVL_CONST：ST_* *)
    iPhase          : INT := 0;        (* 当前任务内阶段（任务模块上报） *)
    iBlockReason    : INT := 0;        (* 阻塞原因码 *)
    iWorkMode       : INT := 0;        (* 工作模式 1=调理 2=治疗 3=老化 *)
    iUserRole       : INT := 0;        (* 角色镜像（HMI 线协议：0=操作员 1=工程师） *)

    (*--- 安全（SAFETY_MANAGER 单写） ---*)
    bHardEstop      : BOOL;            (* 硬急停：断使能（物理链断开 或 锁存升级） *)
    bSoftEstop      : BOOL;            (* 软急停：受控减速 *)
    bSafetyStop     : BOOL;            (* 安全链触发的停止请求（硬/软/保护停机任一） *)
    bProtStop       : BOOL;            (* 保护停机锁存（超力/致命保护，受控减速后锁死，需手动复位） *)
    bHardEstopLatch : BOOL;            (* 硬急停锁存（软急停超时升级；物理链恢复+复位才解除） *)
    bAllAxesIdle    : BOOL;            (* 全轴静止 *)
    bAllAxesRef     : BOOL;            (* 全轴参考有效 *)
    bAllAxesAtInit  : BOOL;            (* 全轴在初始位 *)

    (*--- I/O 镜像（INPUT_ADAPTER 单写，去抖后） ---*)
    ioEstopOK       : BOOL;            (* 急停链路正常（双通道常闭闭合 + 安全继电器未动作） *)
    ioEstop1        : BOOL;            (* 急停通道1 去抖态（X2 常闭，TRUE=闭合正常） *)
    ioEstop2        : BOOL;            (* 急停通道2 去抖态（X3 常闭，TRUE=闭合正常） *)
    ioResetBtn      : BOOL;            (* 复位按钮（X7 去抖） *)
    ioPusherOrigin  : BOOL;            (* 推杆原点（X5 去抖） *)

    (*--- 推杆位置反馈镜像（INPUT_ADAPTER 单写） ---*)
    (* 真实推杆为开关型电推杆，无 AD：位置由 HC_Counter 高速计数器读得，单位 mm；
       角度由 FB_PusherControl 用 GVL_CONST 几何常量（垂直/平行/倾斜偏置/固定角/补偿）
       经余弦定理/ACOS 解算。 *)
    rPusherPosMm    : REAL;            (* 当前推杆位置（mm，HC_Counter.Position） *)
    bPusherPosValid : BOOL;            (* 位置有效（HC_Counter.Valid，无 Error） *)

    (*--- 命令脉冲位（INPUT_ADAPTER 单写，本扫有效） ---*)
    (* H5U 全局变量不支持功能块实例：R_TRIG 在 PRG_InputAdapter 局部 VAR 声明，
       其 .Q 每扫写入下列 BOOL 位；下游直接读位，边沿仅存活一个扫描周期。 *)
    trigStart       : BOOL;            (* S1 启动流程（本扫脉冲） *)
    trigChengJiao   : BOOL;            (* S2 开始成角（本扫脉冲） *)
    trigAllow       : BOOL;            (* S3 确认（本扫脉冲） *)
    trigStop        : BOOL;            (* 停止（本扫脉冲） *)
    trigReset       : BOOL;            (* 复位错误（本扫脉冲） *)
    trigSkipAngle   : BOOL;            (* 跳过成角（本扫脉冲） *)
    (* 电平命令（直接镜像，下游读 .Q 无意义，读电平位） *)
    bPauseLevel     : BOOL;            (* 暂停（电平，Condition.Cmd 或 Sys.Cmd 任一按下） *)
    bResumeLevel    : BOOL;            (* 恢复（电平，Condition.Cmd 或 Sys.Cmd 任一按下） *)
    bFootSignal     : BOOL;            (* 脚踏（电平/脉冲按模式） *)

    (*--- 系统 Sys.Cmd 脉冲请求位（INPUT_ADAPTER 单写，本扫有效） ---*)
    trigServiceMode     : BOOL;        (* 进入维护模式请求 *)
    trigSysHoming       : BOOL;        (* 回零请求 *)
    trigSysStop         : BOOL;        (* 停止请求 *)
    trigAutoStart       : BOOL;        (* 自动流程启动 *)
    trigCalibrate       : BOOL;        (* 推杆标定流程 *)
    trigSysReset        : BOOL;        (* 复位请求（状态机复位/错误复位） *)
    trigAckError        : BOOL;        (* 确认错误 *)
    trigEmgStop         : BOOL;        (* 软急停请求（D488.9，无条件穿透） *)
    trigInitialize      : BOOL;        (* 初始化请求 *)
    trigSvcMechHome     : BOOL;        (* 维护机械回零 *)
    trigSelfTestConfirm : BOOL;        (* 自检安全确认 *)
    trigSelfTestSkip    : BOOL;        (* 自检跳过步 *)
    trigAllPowerOff     : BOOL;        (* 全轴断电 *)
    trigAllPowerOn      : BOOL;        (* 全轴上电 *)
    trigStartSelfTest   : BOOL;        (* 启动自检 *)
    trigServiceDone     : BOOL;        (* 维护完成 *)
    trigReadyCheck      : BOOL;        (* 就绪检查请求 *)
    trigQuickStart      : BOOL;        (* 快速启动（需资格位） *)
    trigForceSkipST     : BOOL;        (* 强制跳过自检（需资格位） *)
    trigClearZeroRetain : BOOL;        (* 清除建零 Retain（6 重门控） *)
    trigLearnBias       : BOOL;        (* 学习冲击轴扭矩基线 *)

    (*--- 系统电平命令镜像（按住有效，离态自动回落） ---*)
    bServiceAuthConfirm : BOOL;        (* 维护授权确认（电平，建零门控） *)
    bNoLoadConfirm      : BOOL;        (* 无负载确认（电平，建零门控） *)
    bRevalidateParams   : BOOL;        (* 参数重校验（电平，P5 消费） *)

    (*--- 三轴命令：[1..3]=Chest冲击/Seat扭角/Leg转角（与 HMI 块轴 ID 对齐，
          见 GVL_CONST AXIS_ID_*）；第二维见 AXCMD_* 索引。INPUT_ADAPTER 单写。 ---*)
    axisPulse       : BOOL[1..3, 1..8];   (* 脉冲命令位（AXCMD_RESET..AXCMD_REQ_DISABLE） *)
    axisEnableReq   : BOOL[1..3];         (* bEnable 电平：请求伺服上电（POWER 消费） *)
    axisJogPos      : BOOL[1..3];         (* bJogPos 正向点动（电平，按住有效） *)
    axisJogNeg      : BOOL[1..3];         (* bJogNeg 负向点动（电平，按住有效） *)
    axisPowerEnable : BOOL[1..3];         (* 伺服使能电平：POWER 单写（分时上电/急停切断），OUTPUT_ADAPTER 只读 *)

    (*--- 电推杆（尾板 TailTilt）命令：INPUT_ADAPTER 单写 ---*)
    trigPushStop        : BOOL;        (* 推杆停止（脉冲） *)
    trigPushReset       : BOOL;        (* 推杆复位（脉冲） *)
    trigPushCalibrate   : BOOL;        (* 推杆标定（脉冲） *)
    trigPushAutoMove    : BOOL;        (* 推杆自动定位（脉冲） *)
    trigPushHome        : BOOL;        (* 推杆回零（脉冲） *)
    trigPushPreset      : BOOL;        (* 推杆手动清零 Preset（脉冲） *)
    trigPushResetError  : BOOL;        (* 推杆清故障（脉冲） *)
    pushEnableReq       : BOOL;        (* 推杆使能（电平） *)
    jogPushUp           : BOOL;        (* 推杆正向上行点动（电平，按住有效） *)
    jogPushDown         : BOOL;        (* 推杆反向下行点动（电平，按住有效） *)

    (*--- P9 建零/标定 Retain 跨环握手（锁存位，不入 CmdPreclear 清扫表） ---*)
    (* TASK_RUNNER 环7 建零成功置 bZeroCommSetReq[i]；PARAM_SERVICE 环8 当扫消费
       写 retainZeroComm[i]:=TRUE 并清请求。推杆标定：fbPusher.bCalibDone 环10 产生，
       OUTPUT_ADAPTER 置 bPushCalibDoneLatch，PARAM_SERVICE 次扫环8 消费写
       retainTailZeroComm:=TRUE 并清。trigClearZeroRetain 环2 脉冲由 PARAM_SERVICE
       环8 消费清全部建零 Retain。 *)
    bZeroCommSetReq     : BOOL[1..3];     (* 三轴建零置位请求（锁存） *)
    bPushCalibDoneLatch : BOOL;           (* 推杆标定完成锁存（跨环） *)

    (*--- 故障提交区（任务模块写 gFaultSubmit，ERROR_MANAGER 唯一消费） ---*)
    gFaultSubmit    : BOOL;            (* 提交脉冲：填好下列字段后置 TRUE *)
    gFaultLevel     : INT;             (* 0=L0 Info 1=L1 Warning 2=L2 Critical *)
    gFaultCode      : INT;             (* 错误码（见 GVL_CONST 段位约定） *)
    gFaultSource    : INT;             (* 来源模块码 *)
    gFaultSubCode   : INT;             (* 子码：轴 9xxx / 驱动器 Er.xxx *)
    gFaultVal1      : INT;             (* 附加值 1 *)
    gFaultVal2      : INT;             (* 附加值 2 *)

    (*--- 扫描监控 ---*)
    (* 看门狗为 BOOL（H5U 内联 TONR 的 Q=> 输出），上移为全局 mnTScanWatchdog（见下方 PRG_Main 分组） *)
    diScanCount     : DINT;            (* 扫描计数（心跳，任务组态按 10ms；超时/持续计时基准） *)
    diMsTick        : DINT;            (* 毫秒运行刻度（上电起 ms，MONITOR 每扫 +扫描周期）：事件时间戳源。
                                          非真实日历时钟；日志若需年月日时分秒，待现场引入 RTC 库 FB
                                          （InoProShop 平台符号以现场库为准，离线不臆造）后再替换。 *)

    (*--- 运行统计累计器（P11，HmiOutput 写入 Sys.Runtime；非保持，上电清零） ---*)
    diStatAgingCycles : DINT;          (* 老化循环累计（老化批完成 +目标循环数） *)
    diStatTotalCycles : DINT;          (* 总循环累计（任一模式每完成 16 段循环表 +1） *)
    diStatRunTime     : DINT;          (* 自动流程累计运行时长（ms；暂停不计时） *)

    (*========================================================================
      POU 私有工作变量（H5U 编辑器不允许 PRG/FC 声明局部简单变量，
      故全部上移为全局；按所属 POU 加前缀分组，仅该 POU 读写。
      功能块实例 / TRIG.R_TRIG 边沿实例仍保留在各 POU 局部 VAR。）
      ========================================================================*)

    (*--- PRG_CmdPreclear（环1 命令清扫） ---*)
    cpIAxis  : INT;                    (* 轴清扫循环下标 1..3 *)
    cpICmd   : INT;                    (* 轴脉冲位循环下标 1..AXCMD_MAX *)

    (*--- PRG_InputAdapter（环2 输入适配） ---*)
    iaTEstop1Db    : BOOL;             (* 急停通道1 去抖输出（X2 常闭，内联 TONR Q=>） *)
    iaTEstop2Db    : BOOL;             (* 急停通道2 去抖输出（X3 常闭） *)
    iaTSafeRelayDb : BOOL;             (* 安全继电器去抖输出（X4 常开） *)
    iaTOriginDb    : BOOL;             (* 推杆原点传感器去抖输出（X5） *)
    iaTResetDb     : BOOL;             (* 复位按钮去抖输出（X7） *)
    iaTDbTime      : TIME := T#30MS;   (* 去抖时间常数（内联 TONR PT） *)
    iaDiHscPos     : DINT;             (* HC_Counter.Position 原始位置（mm，DINT） *)
    iaBHscValid    : BOOL;             (* HC_Counter.Valid *)
    iaBHscError    : BOOL;             (* HC_Counter.Error *)
    iaWHscErrId    : WORD;             (* HC_Counter.ErrorID *)

    (*--- PRG_ErrorManager（环4 故障管理） ---*)
    emIPos     : INT;                  (* 队列游标（兼容保留） *)
    emTWarnAge : BOOL;                 (* 警告存活计时（内联 TONR Q=>） *)

    (*--- PRG_ModeManager（环5 模式管理） ---*)
    mmBEngineer : BOOL;                (* 工程师门：角色=工程师 且 权限码=16#5A *)
    mmBReadyAll : BOOL;                (* 六项资格全具备 *)
    mmDiMask    : DINT;                (* 资格掩码（位置位=缺项） *)
    mmIWarnDv   : INT;                 (* 就绪不齐 Warning 提交节流（扫计数） *)

    (*--- PRG_SafetyManager（环6 安全管理） ---*)
    smTMismatch      : BOOL;           (* 双通道不一致去抖（Q=>） *)
    smBSoftStopActive: BOOL;           (* 软急停减速停车电平（停稳滑行后自动解除） *)
    smDiSoftDecelCnt : DINT;           (* 停车电平有效但轴未全静止计数（×10ms，≥500 升级硬急停） *)
    smDiCoastCnt     : DINT;           (* 软急停停稳后滑行计数（达 diEmergencyCoastMs 解除） *)
    smBHardPhysical  : BOOL;           (* 物理硬急停态（去抖，排除锁存升级） *)
    smBChanMismatch  : BOOL;           (* 急停双通道不一致（去抖前） *)
    smBAnyEncoderFlt : BOOL;           (* 任一轴编码器故障 *)
    smBAnyHwLimit    : BOOL;           (* 任一轴硬限位触发 *)
    smBAnyOverForce  : BOOL;           (* 任一轴超力锁存/实时超力 *)

    (*--- PRG_ParamService（环8 参数服务） ---*)
    psIMac0  : INT;                    (* MAC 承接第1字节（_Ethernet.MACAddress 为 USINT，截低 8 位） *)
    psIMac1  : INT;                    (* MAC 承接第2字节 *)
    psIMac2  : INT;                    (* MAC 承接第3字节 *)
    psBVC    : BOOL;                   (* 校验通过（FC_ValidateParams 输出承接） *)
    psIVCode : INT;                    (* 校验错误码 *)
    psIVAxis : INT;                    (* 错误轴 *)
    psIVField: INT;                    (* 错误字段 *)
    psI      : INT;                    (* 通用循环索引 *)

    (*--- PRG_TaskRunner（环7 任务运行） ---*)
    trIPrevState    : INT;             (* 上扫 iState（进入沿判定） *)
    trBStateEntry   : BOOL;            (* 本扫为新状态首扫 *)
    trIStepHom      : INT;             (* 普通回零步（HOMSEQ_*） *)
    trIStepEmh      : INT;             (* 紧急回零步（EMH_*） *)
    trIStepSt       : INT;             (* 自检步（ST_GATE..ST_STEP_FAIL） *)
    trIStepCal      : INT;             (* 建零步（CAL_*） *)
    trDiSnap        : DINT;            (* 任务级起始扫描快照（超时判定） *)
    trIAxis         : INT;             (* 当前活动轴下标 1..3 *)
    trBAxisDone     : BOOL[1..3];      (* 各轴任务完成（到位+静止+在初始位） *)
    trRInit         : REAL[1..3];      (* 各轴初始位镜像（runAxis[i].rInitPos） *)
    trRJogV         : REAL[1..3];      (* 各轴 Jog 主速镜像（runHoming） *)
    trRCrawlV       : REAL[1..3];      (* 各轴爬行速镜像 *)
    trRApproach     : REAL[1..3];      (* 各轴接近区镜像 *)
    trRHyst         : REAL[1..3];      (* 各轴到位迟滞镜像 *)
    trIRetry        : INT[1..3];       (* 各轴防夹重试计数 *)
    trIEmhAxis      : INT;             (* 紧急回零活动轴下标 1..3 *)
    trDiPinchSnap   : DINT;            (* 防夹撤力等待快照 *)
    trBDirtyAxis    : BOOL;            (* 脏1：三轴活动故障 *)
    trBDirtyForce   : BOOL;            (* 脏2：超力锁存/保护停机 *)
    trBDirtyPusher  : BOOL;            (* 脏3：推杆传感器异常 *)
    trBDirtyParam   : BOOL;            (* 脏4：参数需重校验 *)
    trIStAxis       : INT;             (* 自检摆动当前轴 1..3 *)
    trIStPhase      : INT;             (* 单轴摆动相位 0=+2° 1=-2° 2=归位 *)
    trDiStSnap      : DINT;            (* 自检单段快照 *)
    trDiStGlobalSnap: DINT;            (* 自检全局快照 *)
    trDiPushSnap    : DINT;            (* 推杆校准/成角快照 *)
    trBSelfTestSkipped: BOOL;          (* 本次自检经跳过/强跳完成 *)
    trDiCalSnap     : DINT;            (* 建零命令发出快照（Retain 回读超时） *)
    trBFaultLat     : BOOL;            (* 有未消费故障锁存 *)
    trBFaultSent    : BOOL;            (* 锁存故障已装填 gFaultSubmit *)
    trILatSentCode  : INT;             (* 已提交的故障码（锁存期换码则重发） *)
    trILatLevel     : INT;             (* 锁存故障级别 *)
    trILatCode      : INT;             (* 锁存故障码 *)
    trILatSource    : INT;             (* 锁存故障源 *)
    trILatSub       : INT;             (* 锁存故障子码 *)
    trBEmhPinch     : BOOL;            (* 活动轴净扭矩超阈（防夹） *)
    trBEmhAtInit    : BOOL;            (* 活动轴进入到位迟滞窗口 *)
    trIStepCond     : INT;             (* 调理步号 105..900（CONDSEQ_*） *)
    trIStepStop     : INT;             (* 停止降落步号 6000/6010（STOPSEQ_*） *)
    trICondCycle    : INT;             (* 当前循环计数（1 起） *)
    trICondTarget   : INT;             (* 目标循环数（runCond.iCycleCount） *)
    trDiCondBatch   : DINT;            (* 当前批次（1 起，老化） *)
    trDiCondSnap    : DINT;            (* 单批起始快照（总超时判定） *)
    trDiBatchSnap   : DINT;            (* 批间等待快照 *)
    trDiConfirmSnap : DINT;            (* 108/120 等待确认快照 *)
    trDiCondDoneSnap: DINT;            (* 三轴完成去抖快照 *)
    trBCondPaused   : BOOL;            (* 130 暂停态 *)
    trBAgingAuto    : BOOL;            (* 本任务为老化（WORKMODE_AGING 快照） *)
    trBAutoSignal   : BOOL;            (* 老化内部自动信号位 *)
    trBCondAngleSkip: BOOL;            (* 本批跳过成角（trigSkipAngle） *)
    trBCondCnfTout  : BOOL;            (* 确认超时 7007 已上报 *)
    trBCondRunStart : BOOL;            (* 130 循环启动锁存 *)

    (*--- PRG_OutputAdapter（环10 输出适配） ---*)
    oaISel : INT;                      (* 本扫选中的故障源（0=无 1..3=轴 4=推杆） *)

    (*--- PRG_Power（环9 上电时序） ---*)
    pwIPwrStep  : INT := 0;            (* 0=全断 1=Chest使能 2=Chest等间隔 3=Seat使能 4=Seat等间隔 5=Leg使能 6=全上电完成 *)
    pwBPwrReq   : BOOL;                (* 上电请求锁存 *)
    pwDiStepSnap: DINT;                (* 当前步进入扫描计数 *)
    pwBDisReq   : BOOL[1..3];          (* 单轴断使能请求锁存（AXCMD_REQ_DISABLE 脉冲） *)

    (*--- PRG_Main（主循环/看门狗） ---*)
    mnTScanWatchdog : BOOL;            (* 扫描看门狗超时标志（预留：待绑定 H5U 任务看门狗系统变量；置位时 SAFETY_MANAGER 上报 1007；无应用内 TONR 驱动，详见 PRG_Main 注释） *)

    (*--- FC_ValidateParams（参数校验函数，函数内私有工作变量） ---*)
    vpI   : INT;                       (* 段索引 1..16（FOR 循环） *)
    vpCfg : Stru_AxisLimitConfig;      (* 轴 Config 校验用局部视图 *)
END_VAR

(* ---- GVL_IoMap.st ---- *)
(*============================================================================
  物理 I/O 映射（H5U A8）—— 以 old/变量表/GVL_IoMap.csv（硬件组态导出）为准
  ----------------------------------------------------------------------------
  本机 I/O（CSV 软元件地址）：
    急停双通道：I_Estop1=X2、I_Estop2=X3（均常闭，FALSE=拍下）
    安全继电器：I_SafeRelay=X4（常开，TRUE=拍下）
    复位按钮：I_ResetBtn=X7
    推杆原点：I_PusherOrigin=X5；推杆限位：正/负（未接线，预留无地址）
    推杆输出：Q_Pusher_Up=Y5（上行/正转）、Q_Pusher_Down=Y6（下行/反转）
    推杆位置：开关型电推杆无 AD，位置由 HC_Counter 内联指令高速计数器轴读得
              （单位 mm，Position 直接为 REAL；轴在 H5U 高速计数器组态中定义，
              Axis_电推杆 须与组态轴名逐字一致）
  注：InoProShop 中 X0..X7 ↔ %IX0.0..%IX0.7、Y0..Y7 ↔ %QX0.0..%QX0.7，
      下载后须按硬件组态核对 X/Y 与 %IX/%QX 映射；以下 % 地址由 Xn/Yn 推出。
  EtherCAT：3× M900 伺服轴引用 Axis_胸背/臀盘/臀腿在 H5U 配置文件（设备树）
      中已定义为全局变量，CSV 变量表不含；此处保留声明供 MC 指令引用，
      组态轴名须与这三个标识符逐字一致。
==========================================================================*)
VAR_GLOBAL
    (*--- 数字量输入（去抖在 INPUT_ADAPTER 完成） ---*)
    I_Estop1       AT %IX0.2 : BOOL;   (* 物理急停通道1（X2，常闭：FALSE=拍下） *)
    I_Estop2       AT %IX0.3 : BOOL;   (* 物理急停通道2（X3，常闭：FALSE=拍下） *)
    I_SafeRelay    AT %IX0.4 : BOOL;   (* 安全继电器（X4，常开：TRUE=拍下） *)
    I_PusherOrigin AT %IX0.5 : BOOL;   (* 电推杆原点传感器（X5） *)
    I_ResetBtn     AT %IX0.7 : BOOL;   (* 复位按钮（X7） *)
    I_PusherPosLim           : BOOL;   (* 推杆正限位（未接线，预留） *)
    I_PusherNegLim           : BOOL;   (* 推杆负限位（未接线，预留） *)

    (*--- 数字量输出 ---*)
    Q_Pusher_Up    AT %QX0.5 : BOOL;   (* 推杆上行/正转（Y5），方向取反由 Config 决定 *)
    Q_Pusher_Down  AT %QX0.6 : BOOL;   (* 推杆下行/反转（Y6） *)

    (*--- EtherCAT 总线：3× M900 伺服（CiA402）轴引用（H5U 配置文件已定义，此处保留） ---*)
    Axis_胸背      : AXIS_REF;         (* 冲击轴（ChestImpact） *)
    Axis_臀盘      : AXIS_REF;         (* 扭角轴（SeatTwist）  *)
    Axis_臀腿      : AXIS_REF;         (* 转角轴（LegAngle）   *)

    (*--- 高速计数器轴：尾板推杆位置反馈（H5U 高速计数器组态已定义，HC_Counter 内联引用；
          Position 直接为 REAL，单位 mm；轴名须与组态逐字一致） ---*)
    Axis_电推杆    : AXIS_REF;         (* 推杆位置计数轴（TailTilt，mm） *)
END_VAR

(* ---- GVL_Params.st ---- *)
(*============================================================================
  GVL_Params —— 参数三区模型（P5）
  ----------------------------------------------------------------------------
  三区：
    编辑缓冲 = HMI D 区（HMI.Condition.Param / 各轴 .Config / HomingParams.Params /
               TailTilt.Config），HMI 直接读写，Apply 前不影响运行。
    运行区   = 本 GVL 的 run*（非保持），任务/运动 FB 只读本区；Apply 校验通过后
               由编辑缓冲覆盖；上电从 Retain 区装载，Retain 无效则用工厂默认。
    Retain区 = 本 GVL 的 retain*（VAR_GLOBAL RETAIN，断电保持），Save 时由运行区
               写入；含建零标志 bZeroCommissioned。
  单写源：本 GVL 全部变量仅 PRG_ParamService 可写，其余程序只读 run*。
  轴数组下标与全局约定一致（H5U base 0）：0=ChestImpact 冲击 / 1=SeatTwist 扭角 / 2=LegAngle 转角。
==========================================================================*)
VAR_GLOBAL
    (*--- 运行区（生效值，任务读） ---*)
    runCond             : Stru_CondParams;          (* 调理参数运行区 *)
    runAxis             : Stru_AxisLimitConfig[3];  (* 三轴限位/运动配置运行区，下标 0=Chest 1=Seat 2=Leg *)
    runHoming           : Stru_HomingParams;        (* 回零参数运行区 *)
    runPusher           : Stru_PusherLimitConfig;   (* 推杆配置运行区 *)
    bRunParamValid      : BOOL;                     (* 运行区参数已成功 Apply（快照有效） *)

    (*--- 上电初始化标志（非保持，每次下载/上电首扫 FALSE） ---*)
    bParamBootDone      : BOOL;
END_VAR

VAR_GLOBAL RETAIN
    (*--- Retain 区（断电保持，Save 时写入） ---*)
    retainValid         : BOOL;                     (* Retain 区有效标志（首板为 FALSE→装默认） *)
    retainCond          : Stru_CondParams;          (* 调理参数保持区 *)
    retainAxis          : Stru_AxisLimitConfig[3];  (* 三轴配置保持区，下标 0..2 *)
    retainHoming        : Stru_HomingParams;       (* 回零参数保持区 *)
    retainPusher        : Stru_PusherLimitConfig;   (* 推杆配置保持区 *)
    retainZeroComm      : BOOL[3];                  (* 三轴建零标志 bZeroCommissioned（工厂建零后置位），下标 0..2 *)
    retainTailZeroComm  : BOOL;                     (* 推杆参考/标定保持标志 bCalibrated *)
    retainDeviceNo      : DINT;                     (* 设备编号保持区（工厂烧录/维护 Apply 写入） *)
END_VAR
